# EPICS substitutions: vaccelApp/Db/offset.substitutions
file db/offset.rec
{
	pattern{ ELEMENT }
               { q1m1d1r }

}
